ORGANIZATION_BLOCK MAIN:OB1
TITLE=程序注释
BEGIN
Network 1
//  程序段注释
LD     SM0.1
S      M2.0, 1
Network 2
LD     M2.0
S      Q0.0, 1
TON    T37, 10
A      T37
R      M2.0, 1
S      M2.1, 1
Network 3
LD     M2.1
S      Q0.1, 1
TON    T38, 20
A      T38
R      M2.1, 1
S      M2.0, 1
END_ORGANIZATION_BLOCK
SUBROUTINE_BLOCK SBR_0:SBR0
TITLE=子程序注释
BEGIN
Network 1
//  程序段注释
END_SUBROUTINE_BLOCK
INTERRUPT_BLOCK INT_0:INT0
TITLE=中断例程注释
BEGIN
Network 1
//  程序段注释
END_INTERRUPT_BLOCK
